// TIA Portal V20 export
TYPE "typeSequenceControlNodeConveyorJobInterface"
// stored: Namespace Unit1.Em7
   STRUCT
      commands : "Unit1.Em7.typeSequenceControlNodeConveyorJobInterfaceCommands";
      monitoring { S7_SetPoint := 'True'} : "Unit1.Em7.typeSequenceControlNodeConveyorJobInterfaceMonitoring";
   END_STRUCT;
END_TYPE
